Universal Robots PolyScope program: position.urp

Program position (installation=default directory=/programs createdIn=5.2.0.61336 lastSavedIn=5.2.0.61336 robotSerialNumber=20195500451)
Calibrated DH parameters: a=[0.00002, -0.231658, -0.317125, 0.000011, 0.000055, 0]; d=[0.162082, 123.190176, -180.284242, 57.22734, 0.099524, 0.09934]; alpha=[1.569304, 0.00289, 0.004025, 1.569925, -1.569026, 0]; deltaTheta=[0, 0.993923, 4.662183, 0.627072, 0.000001, 0]
Robot Program (runOnlyOnce=false)
  MoveJ speed 60 deg/s, acceleration 80 deg/s^2 (useActiveTCP=true) feature=Base
    Waypoint Waypoint_1: motionParameters(nextMotionTime=1 blendRadius=0.05); TCP in base x=224.186 y=-61.012 z=1078.412 mm, rx=-1.0701 ry=1.4002 rz=-1.4035 rad; joints [75.057, -90.002, 0, -90, 0, 0.002] deg
    Waypoint Waypoint_3: motionParameters(nextMotionTime=1 blendRadius=0.028); TCP in base x=112.8 y=203.121 z=1078.412 mm, rx=-1.5318 ry=0.3965 rz=-0.3973 rad; joints [151.259, -89.997, 0.001, -90, -0.002, 0.003] deg
